// TIA Portal V17 export
// export: Created 2025-07-17T00:36:38.5858719Z, ExportSetting WithDefaults, DisplayName Totally Integrated Automation Portal, DisplayVersion V17, DisplayName TIA Portal Openness, DisplayVersion V17, DisplayName TIA Portal Version Control Interface, DisplayVersion V17, DisplayName STEP 7 Professional, DisplayVersion V17, DisplayName STEP 7 Safety, DisplayVersion V17, DisplayName WinCC Advanced / Unified PC, DisplayVersion V17
FUNCTION "tank_level" : Void   // FC3, LAD
{ S7_Optimized_Access := 'TRUE' }
VERSION : 0.1
// stored: AutoNumber true, IsIECCheckEnabled false, SetENOAutomatically false, UDAEnableTagReadback false
   VAR_TEMP
      tank_level_temp1 : Real;
      tank_level_temp2 : Real;
   END_VAR
BEGIN

REGION Network 1
   // 读取罐液罐液位
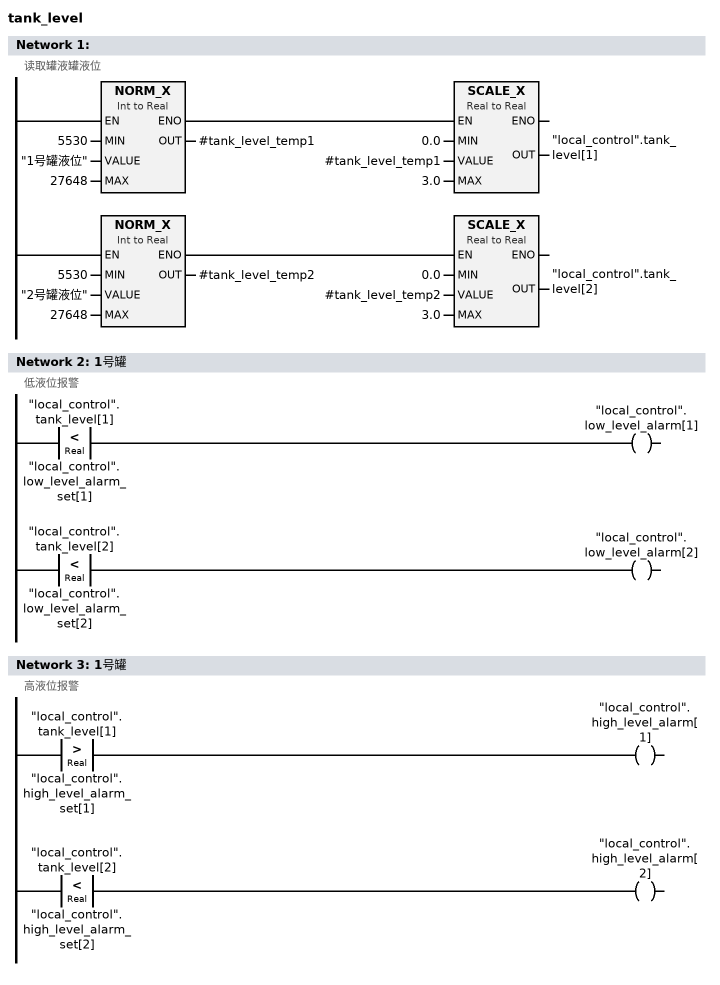
   RUNG wire#powerrail
      { S7_Templates := "[SrcType := Int, DestType := Real]" } Normalize(min := 5530, value := "1号罐液位", max := 27648, out => #tank_level_temp1)
      { S7_Templates := "[SrcType := Real, DestType := Real]" } Scale(min := 0.0, value := #tank_level_temp1, max := 3.0, out => "local_control".tank_level[1])
   END_RUNG
   RUNG wire#powerrail
      { S7_Templates := "[SrcType := Int, DestType := Real]" } Normalize(min := 5530, value := "2号罐液位", max := 27648, out => #tank_level_temp2)
      { S7_Templates := "[SrcType := Real, DestType := Real]" } Scale(min := 0.0, value := #tank_level_temp2, max := 3.0, out => "local_control".tank_level[2])
   END_RUNG
   // the same network as SCL:
   #tank_level_temp1 := NORM_X(MIN := 5530, VALUE := "1号罐液位", MAX := 27648);
   "local_control".tank_level[1] := SCALE_X(MIN := 0.0, VALUE := #tank_level_temp1, MAX := 3.0);
   #tank_level_temp2 := NORM_X(MIN := 5530, VALUE := "2号罐液位", MAX := 27648);
   "local_control".tank_level[2] := SCALE_X(MIN := 0.0, VALUE := #tank_level_temp2, MAX := 3.0);
END_REGION

REGION Network 2: 1号罐
   // 低液位报警
   RUNG wire#powerrail
      { S7_Templates := "SrcType := Real" } LT_Contact(in1 := "local_control".tank_level[1], in2 := "local_control".low_level_alarm_set[1])
      Coil( "local_control".low_level_alarm[1] )
   END_RUNG
   RUNG wire#powerrail
      { S7_Templates := "SrcType := Real" } LT_Contact(in1 := "local_control".tank_level[2], in2 := "local_control".low_level_alarm_set[2])
      Coil( "local_control".low_level_alarm[2] )
   END_RUNG
   // the same network as SCL:
   "local_control".low_level_alarm[1] := "local_control".tank_level[1] < "local_control".low_level_alarm_set[1];
   "local_control".low_level_alarm[2] := "local_control".tank_level[2] < "local_control".low_level_alarm_set[2];
END_REGION

REGION Network 3: 1号罐
   // 高液位报警
   RUNG wire#powerrail
      { S7_Templates := "SrcType := Real" } GT_Contact(in1 := "local_control".tank_level[1], in2 := "local_control".high_level_alarm_set[1])
      Coil( "local_control".high_level_alarm[1] )
   END_RUNG
   RUNG wire#powerrail
      { S7_Templates := "SrcType := Real" } LT_Contact(in1 := "local_control".tank_level[2], in2 := "local_control".high_level_alarm_set[2])
      Coil( "local_control".high_level_alarm[2] )
   END_RUNG
   // the same network as SCL:
   "local_control".high_level_alarm[1] := "local_control".tank_level[1] > "local_control".high_level_alarm_set[1];
   "local_control".high_level_alarm[2] := "local_control".tank_level[2] < "local_control".high_level_alarm_set[2];
END_REGION
END_FUNCTION
